TYPE CM_Valve_HMI :
STRUCT
	Start		: BOOL;
	Stop		: BOOL;
	Reset		: BOOL;
	Abort		: BOOL;
	Clear		: BOOL;
	UnSuspend	: BOOL;
	Suspend		: BOOL;
	UnHold		: BOOL;
	Hold		: BOOL;
	Auto		: BOOL;
	Manueel		: BOOL;
	Open		: BOOL;
	Close		: BOOL;
END_STRUCT
END_TYPE

(* stored: Version 1.1.0.1, ProductVersion 3.1.4024.12
   DUT CM_Valve_HMI: Id {455dd156-9e1c-44cf-aa0c-b3c9361a41dd} *)
